(* PLC project Unnamed, Unknown Unnamed 1 *)
(* stored: creationDateTime 2025-12-04T16:18:24, modificationDateTime 2025-12-04T16:18:24 *)

CONFIGURATION Config0
  RESOURCE Res0 ON PLC
  END_RESOURCE
END_CONFIGURATION
